(* PLC project LibIT_DI, lamsystems-it.ru LibIT_DI 1 *)
(* stored: creationDateTime 2019-11-13T09:37:45, productRelease 0, modificationDateTime 2023-02-28T17:02:11, version 1 *)

(* Установка режима работы дискретного входа *)
FUNCTION_BLOCK DIMode
  VAR_INPUT
    Ex : BOOL := FALSE;  (* разрешение на выполнение *)
    DIn : BYTE := 0;  (* номер входа *)
    M : BYTE := 0;  (* режим работы *)
  END_VAR
  VAR_OUTPUT
    Ok : BYTE := 0;  (* код результата исполнения блока *)
  END_VAR

            {extern void App_DIMode(DIMODE*);App_DIMode(data__);}

          
END_FUNCTION_BLOCK

(* Текущий режим и состояние входа DI *)
FUNCTION_BLOCK DIStatus
  VAR_INPUT
    DIn : BYTE := 0;  (* номер входа *)
  END_VAR
  VAR_OUTPUT
    Om : BYTE := 0;  (* режим работы (установленный) *)
    Ok : BYTE := 0;  (* код результата исполнения блока *)
  END_VAR

            {extern void App_DIStatus(DISTATUS*);App_DIStatus(data__);}

          
END_FUNCTION_BLOCK

(* Получить значение нормального дискретного входа *)
FUNCTION_BLOCK DIVal
  VAR_INPUT
    Ex : BOOL := FALSE;  (* разрешение на выполнение *)
    DIn : BYTE := 0;  (* номер входа *)
  END_VAR
  VAR_OUTPUT
    Ov : BOOL := FALSE;  (* значение *)
    Ok : BYTE := 0;  (* код результата исполнения блока *)
  END_VAR

            {extern void App_DIVal(DIVAL*);App_DIVal(data__);}

          
END_FUNCTION_BLOCK

(* Сброс счетного входа или входа тахометра *)
FUNCTION_BLOCK DICntRst
  VAR_INPUT
    Ex : BOOL := FALSE;  (* разрешение на выполнение *)
    DIn : BYTE := 0;  (* номер входа *)
    Rst : BOOL := FALSE;  (* команда сброса *)
  END_VAR
  VAR_OUTPUT
    Ok : BYTE := 0;  (* код результата исполнения блока *)
  END_VAR

            {extern void App_DICntRst(DICNTRST*);App_DICntRst(data__);}

          
END_FUNCTION_BLOCK

(* Получить значение входа тахометра *)
FUNCTION_BLOCK DISetCfgCntT
  VAR_INPUT
    Ex : BOOL := FALSE;  (* разрешение на выполнение *)
    DIn : BYTE := 0;  (* номер входа *)
    Sp : WORD := 0;  (* уставка *)
    EnCmpMd : BOOL := FALSE;  (* разрешение работы по уставке *)
  END_VAR
  VAR_OUTPUT
    Ok : BYTE := 0;  (* код результата исполнения блока *)
  END_VAR

            {extern void App_DISetCfgCntT(DISETCFGCNTT*);App_DISetCfgCntT(data__);}

          
END_FUNCTION_BLOCK

(* Получить значение счетного входа *)
FUNCTION_BLOCK DISetCfgCnt
  VAR_INPUT
    Ex : BOOL := FALSE;  (* разрешение на выполнение *)
    DIn : BYTE := 0;  (* номер входа *)
    Sp : DWORD := 0;  (* уставка *)
    EnCmpMd : BOOL := FALSE;  (* разрешение работы по уставке *)
  END_VAR
  VAR_OUTPUT
    Ok : BYTE := 0;  (* код результата исполнения блока *)
  END_VAR

            {extern void App_DISetCfgCnt(DISETCFGCNT*);App_DISetCfgCnt(data__);}

          
END_FUNCTION_BLOCK

FUNCTION_BLOCK DISetCfgEnc
  VAR_INPUT
    Ex : BOOL := FALSE;  (* разрешение на выполнение *)
    DIn : BYTE := 0;  (* номер первичного группового входа *)
    SpA : DWORD := 0;  (* уставка счетчика фазы A *)
    EnCmpMdA : BOOL := FALSE;  (* разрешение работы счетчика фазы A по уставке *)
    SpB : DWORD := 0;  (* уставка счетчика фазы B *)
    EnCmpMdB : BOOL := FALSE;  (* разрешение работы счетчика фазы B по уставке *)
    SpT : WORD := 0;  (* уставка тахометра *)
    EnCmpMdT : BOOL := FALSE;  (* разрешение работы тахометра по уставке *)
    SpMultiple : BYTE := 0;  (* множитель энкодера *)
  END_VAR
  VAR_OUTPUT
    Ok : BYTE := 0;  (* код результата исполнения блока *)
  END_VAR

            {extern void App_DISetCfgEnc(DISETCFGENC*);App_DISetCfgEnc(data__);}

          
END_FUNCTION_BLOCK

FUNCTION_BLOCK DIStateCfgCntT
  VAR_INPUT
    DIn : BYTE := 0;  (* номер входа *)
  END_VAR
  VAR_OUTPUT
    OSp : WORD := 0;  (* значение уставки *)
    OEnCmpMd : BOOL := FALSE;  (* разрешение работы по уставке *)
    Ok : BYTE := 0;  (* код результата исполнения блока *)
  END_VAR

            {extern void App_DIStateCfgCntT(DISTATECFGCNTT*);App_DIStateCfgCntT(data__);}

          
END_FUNCTION_BLOCK

(* Получить значение счетного входа *)
FUNCTION_BLOCK DIStateCfgCnt
  VAR_INPUT
    DIn : BYTE := 0;  (* номер входа *)
  END_VAR
  VAR_OUTPUT
    OSp : DWORD := 0;  (* значение счетчика *)
    OEnCmpMd : BOOL := FALSE;  (* разрешение работы п уставке *)
    Ok : BYTE := 0;  (* код результата исполнения блока *)
  END_VAR

            {extern void App_DIStateCfgCnt(DISTATECFGCNT*);App_DIStateCfgCnt(data__);}

          
END_FUNCTION_BLOCK

FUNCTION_BLOCK DIStateCfgEnc
  VAR_INPUT
    DIn : BYTE := 0;  (* номер первичного группового входа *)
  END_VAR
  VAR_OUTPUT
    OSpA : DWORD := 0;  (* уставка счетчика фазы A *)
    OEnCmpMdA : BOOL := FALSE;  (* разрешение работы счетчика фазы A по уставке *)
    OSpB : DWORD := 0;  (* уставка счетчика фазы B *)
    OEnCmpMdB : BOOL := FALSE;  (* разрешение работы счетчика фазы B по уставке *)
    OSpT : WORD := 0;  (* уставка тахометра *)
    OEnCmpMdT : BOOL := FALSE;  (* разрешение работы тахометра по уставке *)
  END_VAR
  VAR_INPUT
    SpMultiple : BYTE := 0;  (* множитель энкодера *)
  END_VAR
  VAR_OUTPUT
    Ok : BYTE := 0;  (* код результата исполнения блока *)
  END_VAR

            {extern void App_DIStateCfgEnc(DISTATECFGENC*);App_DIStateCfgEnc(data__);}

          
END_FUNCTION_BLOCK

(* Получить значение входа тахометра *)
FUNCTION_BLOCK DICntT
  VAR_INPUT
    Ex : BOOL := FALSE;  (* разрешение на выполнение *)
    DIn : BYTE := 0;  (* номер входа *)
  END_VAR
  VAR_OUTPUT
    Ov : WORD := 0;  (* значение *)
    OisSet : BOOL := FALSE;  (* признак достижения уставки *)
    Ok : BYTE := 0;  (* код результата исполнения блока *)
  END_VAR

            {extern void App_DICntT(DICNTT*);App_DICntT(data__);}

          
END_FUNCTION_BLOCK

(* Получить значение счетного входа *)
FUNCTION_BLOCK DICnt
  VAR_INPUT
    Ex : BOOL := FALSE;  (* разрешение на выполнение *)
    DIn : BYTE := 0;  (* номер входа *)
  END_VAR
  VAR_OUTPUT
    Ov : DWORD := 0;  (* значение счетчика *)
    OisSet : BOOL := FALSE;  (* признак достижения уставки *)
    Ok : BYTE := 0;  (* код результата исполнения блока *)
  END_VAR

            {extern void App_DICnt(DICNT*);App_DICnt(data__);}

          
END_FUNCTION_BLOCK

(* Получить значения входов счетного энкодера *)
FUNCTION_BLOCK DIEnc
  VAR_INPUT
    Ex : BOOL := FALSE;  (* разрешение на выполнение *)
    DIn : BYTE := 0;  (* номер первичного группового входа *)
  END_VAR
  VAR_OUTPUT
    OvA : DWORD := 0;  (* значение счетчика фазы A *)
    OisSetA : BOOL := FALSE;  (* признак достижения уставки счетчиком фазы A *)
    OvB : DWORD := 0;  (* значение счетчика фазы B *)
    OisSetB : BOOL := FALSE;  (* признак достижения уставки счетчиком фазы B *)
    OvT : WORD := 0;  (* значение тахометра *)
    OisSetT : BOOL := FALSE;  (* признак достижения уставки тахометром *)
    Ok : BYTE := 0;  (* код результата исполнения блока *)
  END_VAR

            {extern void App_DIEnc(DIENC*);App_DIEnc(data__);}

          
END_FUNCTION_BLOCK
